Fanuc TP program (LS listing): aaaj_main.ls

/PROG  AAAJ_MAIN
/ATTR
OWNER		= MNEDITOR;
COMMENT		= "";
PROG_SIZE	= 176;
CREATE		= DATE 20-12-01  TIME 17:56:08;
MODIFIED	= DATE 20-12-01  TIME 21:13:36;
FILE_NAME	= ;
VERSION		= 0;
LINE_COUNT	= 2;
MEMORY_SIZE	= 556;
PROTECT		= READ_WRITE;
TCD:  STACK_SIZE	= 0,
      TASK_PRIORITY	= 50,
      TIME_SLICE	= 0,
      BUSY_LAMP_OFF	= 0,
      ABORT_REQUEST	= 0,
      PAUSE_REQUEST	= 0;
DEFAULT_GROUP	= 1,*,*,*,*;
CONTROL_CODE	= 00000000 00000000;
/APPL
/MN
   1:  CALL AAAJ_HOME    ;
   2:  CALL AAAJ_L123    ;
/POS
/END
